TYPE StructureWithArray :
STRUCT
	myArray : ARRAY [0..2] OF LREAL;
END_STRUCT
END_TYPE

(* stored: Version 1.1.0.1, ProductVersion 3.1.4024.11
   DUT StructureWithArray: Id {e0396530-45b9-49f4-93a8-80c5025244d2} *)
